// TIA Portal V16 export
// export: Created 2023-08-28T09:37:53.7416851Z, ExportSetting WithDefaults, DisplayName Totally Integrated Automation Portal, DisplayVersion V16 Update 6, DisplayName TIA Portal Version Control Interface, DisplayVersion V16 Update 2, DisplayName TIA Portal Openness, DisplayVersion V16 Update 6, DisplayName STEP 7 Professional, DisplayVersion V16 Update 6, DisplayName STEP 7 Safety, DisplayVersion V16, DisplayName WinCC Advanced, DisplayVersion V16 Update 6
VAR_GLOBAL   // PLC tag table "Default tag table"
   System_Byte AT %MB1 : Byte;
   FirstScan AT %M1.0 : Bool;
   DiagStatusUpdate AT %M1.1 : Bool;
   AlwaysTRUE AT %M1.2 : Bool;
   AlwaysFALSE AT %M1.3 : Bool;
   Clock_Byte AT %MB2 : Byte;
   Clock_10Hz AT %M2.0 : Bool;
   Clock_5Hz AT %M2.1 : Bool;
   "Clock_2.5Hz" AT %M2.2 : Bool;
   Clock_2Hz AT %M2.3 : Bool;
   "Clock_1.25Hz" AT %M2.4 : Bool;
   Clock_1Hz AT %M2.5 : Bool;
   "Clock_0.625Hz" AT %M2.6 : Bool;
   "Clock_0.5Hz" AT %M2.7 : Bool;
   Byte_Wekt_DRV01_R AT %MB6 : SInt;   // Bytewejściowy Status napędu
   Byte_Wekt_DRV_Temp AT %MB7 : SInt;   // Byte temp pomocniczy przy wyliczeniu wektora
   "DRV01-Bit_A/M" AT %M6.7 : Bool;   // BIt IN statusu napędu Bit Aut/manual (aut=1, manu=0)
   "DRV01-Bit_REM" AT %M6.2 : Bool;   // Bit IN statusu napędu Bit-REM Tryb aut=1 rem=0 (REM sterowanie remontowe)
   "DRV01-Bit_A" AT %M6.0 : Bool;   // Bit IN status napędu Bit-A (Alarm)
   "DRV01-Bit_Z" AT %M6.5 : Bool;   // Bit IN statusu napędu Bit-Z rozkaz załącz
   "DRV01-Bit_W" AT %M6.4 : Bool;   // Bit IN status napędu Bit-W rozkaz wyłącz
   "DRV01-Bit_R" AT %M6.6 : Bool;   // Bit IN status napędu Bit-R sygnał RESET Alarmu
   Byte_Wekt_DRV01_L AT %MB8 : Byte;   // Byte OUT wektor napędu
   Bit_DRV01_A AT %M8.0 : Bool;   // Bit OUT wektor napędu Bit-A Alarm
   Bit_DRV01_REM AT %M8.2 : Bool;   // Bit OUT wektor napędu Bit-REM tryb pracy aut=1 rem=0 (REM-sterowanie remontowe)
   Bit_DRV01_Run AT %M8.3 : Bool;   // Bit OUT wektor napędu Bit-Run (Praca stycznik załączony)
   Bit_DRV01_W AT %M8.4 : Bool;   // Bit OUT wektor napędu Bit-W rozkaz wyłącz
   Bit_DRV01_Z AT %M8.5 : Bool;   // Bit OUT wektor napędu Bit-Z rozkaz załącz
   Bit_DRV01_R AT %M8.6 : Bool;   // Bit OUT wektor napędu Bit-R ( reset alarmu)
   "Bir_DRV01_A/M" AT %M8.7 : Bool;   // Bit OUT wektor napędu Bit-A/M rodzaj pracy auto / manual (aut=1, manu=0)
   Memeory_ResAut AT %M13.2 : Bool;   // Pamięć zbocza resetu bitu automat
   apx AT %MD28 : Real;
   apx1 AT %MD32 : Real;
   apy1 AT %MD24 : Real;
   osx AT %MD50 : Real;
   osx1 AT %MD54 : Real;
   osx2 AT %MD58 : Real;
   osy AT %MD62 : Real;
   osy1 AT %MD66 : Real;
   osy2 AT %MD70 : Real;
   State_PID1 AT %MW74 : Int;
   Error_State_PID1 AT %MD76 : DWord;
   SetpointLimit_H_PID1 AT %M14.0 : Bool;   // Wartość zadanaograniczenie górnego PID1
   SetpointLimit_L_PID1 AT %M14.1 : Bool;   // Wartość zadanaograniczenie dolnego PID1
   InputWarning_H_PID1 AT %M14.2 : Bool;   // Wejście ostrzegawcze progu górnrgo PID1
   InputWarning_L_PID1 AT %M14.3 : Bool;   // Wejście ostrzegawcze progu dolnego PID1
   My_1Hz AT %M206.7 : Bool;   // Generator 1hz
   memK1 AT %M15.1 : Bool;   // Flaga pamięci K1
   pause_1 AT %M15.4 : Bool;   // Dla pomiaru nr 1 funkcji FB3
   pause_2 AT %M15.5 : Bool;   // Pałza dla pomiaru nr 2 funkcji FB3
   "Q1.1" AT %Q1.1 : Bool;
   ProcessMemory_Static_1_setChanging AT %M206.4 : Bool;   // Znacznik pobierania konfiguracji do instancji pamięci peocesu
   Tag_2 AT %MW221 : Int;
   Tag_5 AT %M10101.0 : Bool;
   Reset_symulowany AT %M1040.0 : Bool;   // Pomocniczy w razie symulacji
   Tag_6 AT %M1040.5 : Bool;
   Tag_7 AT %M1040.6 : Bool;
   Tag_8 AT %M1040.7 : Bool;
   sim_ON_OFF_AQ_Falownik AT %M1040.2 : Bool;   // Do symulacji i testów
   Sumul_OnOFF_manual_PID AT %M1100.1 : Bool;
   Symula_K2_OFF_ONN AT %M1100.3 : Bool;   // Do testów
   ResetDodtkowe AT %M1100.6 : Bool;   // Potrzeby testowe
   SymulPomoc_04 AT %M1100.4 : Bool;
   SymulPomoc_05 AT %M1100.5 : Bool;
   "I0.0" AT %I0.0 : Bool;
   "Q0.0" AT %Q0.0 : Bool;
   "Q0.1" AT %Q0.1 : Bool;
   "Q0.2" AT %Q0.2 : Bool;
   "I0.1" AT %I0.1 : Bool;
   "I0.2" AT %I0.2 : Bool;
   "I0.5" AT %I0.5 : Bool;
   "I0.6" AT %I0.6 : Bool;
   "I0.7" AT %I0.7 : Bool;
   "I1.0" AT %I1.0 : Bool;
   "I1.1" AT %I1.1 : Bool;
   "I1.2" AT %I1.2 : Bool;
   "Q0.3" AT %Q0.3 : Bool;
   "Q0.4" AT %Q0.4 : Bool;
   "Q0.5" AT %Q0.5 : Bool;
   "I0.3" AT %I0.3 : Bool;
   "I0.4" AT %I0.4 : Bool;
   "I3.7" AT %I3.7 : Bool;
   "I1.3" AT %I1.3 : Bool;
   "I1.5" AT %I1.5 : Bool;
   "I2.1" AT %I2.1 : Bool;
   "I2.0" AT %I2.0 : Bool;
   "Q1.0" AT %Q1.0 : Bool;
   "Q2.3" AT %Q2.3 : Bool;
   "Q2.2" AT %Q2.2 : Bool;
   "I1.4" AT %I1.4 : Bool;
   "Q0.6" AT %Q0.6 : Bool;
   "Q0.7" AT %Q0.7 : Bool;
   "I2.2" AT %I2.2 : Bool;
   "I2.3" AT %I2.3 : Bool;
   "I2.4" AT %I2.4 : Bool;
   "I2.5" AT %I2.5 : Bool;
   "I2.6" AT %I2.6 : Bool;
   "I2.7" AT %I2.7 : Bool;
   "I3.0" AT %I3.0 : Bool;
   "I3.1" AT %I3.1 : Bool;
   "I3.2" AT %I3.2 : Bool;
   "I3.3" AT %I3.3 : Bool;
   "I3.4" AT %I3.4 : Bool;
   "I3.5" AT %I3.5 : Bool;
   "I3.6" AT %I3.6 : Bool;
   "Q2.0" AT %Q2.0 : Bool;
   "Q2.1" AT %Q2.1 : Bool;
   "Q2.4" AT %Q2.4 : Bool;
   "Q2.5" AT %Q2.5 : Bool;
   "Q2.6" AT %Q2.6 : Bool;
   "Q2.7" AT %Q2.7 : Bool;
   "Q3.0" AT %Q3.0 : Bool;
   "Q3.1" AT %Q3.1 : Bool;
   "Q3.2" AT %Q3.2 : Bool;
   "Q3.3" AT %Q3.3 : Bool;
   "Q3.4" AT %Q3.4 : Bool;
   "Q3.5" AT %Q3.5 : Bool;
   "Q3.6" AT %Q3.6 : Bool;
   "Q3.7" AT %Q3.7 : Bool;
   "I4.0" AT %I4.0 : Bool;
   "I4.1" AT %I4.1 : Bool;
   "I4.2" AT %I4.2 : Bool;
   "I4.3" AT %I4.3 : Bool;
   "I4.4" AT %I4.4 : Bool;
   "I4.5" AT %I4.5 : Bool;
   "I4.6" AT %I4.6 : Bool;
   "I4.7" AT %I4.7 : Bool;
   "Q4.0" AT %Q4.0 : Bool;
   "Q4.1" AT %Q4.1 : Bool;
   "Q4.2" AT %Q4.2 : Bool;
   "Q4.3" AT %Q4.3 : Bool;
   "Q4.4" AT %Q4.4 : Bool;
   "Q4.5" AT %Q4.5 : Bool;
   "Q4.6" AT %Q4.6 : Bool;
   "Q4.7" AT %Q4.7 : Bool;
   Tag_3 AT %MW410 : Int;
   Tag_4 AT %MW500 : Int;
   Tag_9 AT %MW502 : Int;
   Tag_10 AT %MD500 : DWord;
   ByteH_Status_P2 AT %MB62 : Byte;   // status napędu
   ByteH_Status_P3 AT %MB64 : Byte;   // staus napędu
   ByteH_Status_P4 AT %MB66 : Byte;   // status napędu
   activePump_P1 AT %M50.4 : Bool;   // aktywna w trybie automat
   activePump_P2 AT %M50.5 : Bool;   // aktywna w trybie automat
   activePump_P3 AT %M50.6 : Bool;   // aktywna w trybie automat
   activePump_P4 AT %M50.7 : Bool;   // aktywna w trybie automat
   PV_PER_bar_modbus AT %MW400 : Int;   // Wartość bar strefa 1
   increase_O2_no1 AT %M15.6 : Bool;   // Znacznik przyrostu wartości bar 1=przyrost, 0= brak przyrostu
   "PV_PER_bar_modbus(1)" AT %MW402 : Int;   // Wartość bar strefa 2
   Tag_1 AT %M212.3 : Bool;
   stopo_dodatkow_1 AT %M15.7 : Bool;   // wyłączenie dodatkowej 1
   ris1_Hz_Calkul_bar AT %M15.2 : Bool;   // Pamięć zbocza narastającego pomiaru 1 dla funkcji FB3
   ris2_Hz_Calkul_bar AT %M15.3 : Bool;   // Pamięć zbocza narastającego nr2 dla funkcji FB3
   "HMI.przeciążenie_falownika" AT %M800.2 : Bool;   // przeciążenie falownika 1
END_VAR
VAR_GLOBAL CONSTANT   // user constants
   CONST_BUFFER_OB82 : USInt := 200;
   CONST_CUREENT2TEMPERATURE_CONVERT : Real := 50.0;
   CONST_Hz_LEVEL : Real := 33.0;
   CONST_ADC_CONVERT : Real := 27648.0;
   CONST_OUTPUT_CAREENT : Real := 20.0;
   "Local~HSC_1(2)" : Hw_Hsc := 258;
   "Local~HSC_2(2)" : Hw_Hsc := 259;
   "Local~HSC_3(2)" : Hw_Hsc := 260;
   "Local~HSC_4(2)" : Hw_Hsc := 261;
   "Local~HSC_5(2)" : Hw_Hsc := 262;
   "Local~HSC_6(2)" : Hw_Hsc := 263;
   "Local~AI2_1" : Hw_SubModule := 264;
   "Local~DI14_DQ10_1" : Hw_SubModule := 265;
   "Local~Pulse_1(2)" : Hw_Pwm := 266;
   "Local~Pulse_2(2)" : Hw_Pwm := 267;
   "Local~Pulse_3(2)" : Hw_Pwm := 268;
   "Local~Pulse_4(2)" : Hw_Pwm := 269;
   DomZabkowska : DB_WWW := 333;
   Temeratura : DB_WWW := 333;
   "Local(2)" : Hw_SubModule := 50;
   "Local~PROFINET_interface_1(2)" : Hw_Interface := 64;
   "Local~PROFINET_interface_1~Port_1(2)" : Hw_Interface := 65;
   "Local~DI_8x24VDC_1(2)" : Hw_SubModule := 270;
   OB_Main : OB_PCYCLE := 1;
   "OB_Cyclic interrupt" : OB_Cyclic := 30;
   OB_Startup : OB_STARTUP := 100;
   "Local(1)" : Hw_SubModule := 50;
   "Local~PROFINET_interface_1(1)" : Hw_Interface := 64;
   "Local~PROFINET_interface_1~Port_1(1)" : Hw_Interface := 65;
   "Local~HSC_1(1)" : Hw_Hsc := 257;
   "Local~HSC_2(1)" : Hw_Hsc := 258;
   "Local~HSC_3(1)" : Hw_Hsc := 259;
   "Local~HSC_4(1)" : Hw_Hsc := 260;
   "Local~HSC_5(1)" : Hw_Hsc := 261;
   "Local~HSC_6(1)" : Hw_Hsc := 262;
   "Local~AI_2_AQ_2_1" : Hw_SubModule := 263;
   "Local~DI_14_DQ_10_1(1)" : Hw_SubModule := 264;
   "Local~Pulse_1(1)" : Hw_Pwm := 265;
   "Local~Pulse_2(1)" : Hw_Pwm := 266;
   "Local~Pulse_3(1)" : Hw_Pwm := 267;
   "Local~Pulse_4(1)" : Hw_Pwm := 268;
   "OB_Main(1)" : OB_PCYCLE := 1;
   "Local~DI_8x24VDC_1(1)" : Hw_SubModule := 269;
   "OB_Startup(1)" : OB_STARTUP := 100;
   "~Port_2" : Hw_Interface := 66;
   "Local~AQ_4x14BIT_1(1)" : Hw_SubModule := 271;
   "~Port_2(1)" : Hw_Interface := 66;
   MS_TO_S : DInt := 1000;
   MS_TO_M : DInt := 60000;   // Pomocnicza zmienna zamiana ms na minuty
END_VAR
